{attribute addProperty BoxType "EK1100-0000-0018"}
{attribute addProperty Id "Beckhoff_EP9xxxEK1122Beckhoff_EP9xxxEK1122_D439D8FD4662582.75A_0023_EP9224_1037_0017EP9224_179A0949162A_0015_EP9128_2021_0019EP9128_179A0949162A_0014_EP9128_1021_0019EP9128_179A0949162A_0012_EP9128_2021_0018EP9128_179A0949162A_0011_EP9128_1021_0018EP9128_179A0949162A_0009_EP9128_2021_0017EP9128_179A0949162A_0008_EP9128_1021_0017EP9128_179A0949162A_0006_EP9128_2021_0016EP9128_179A0949162A_0005_EP9128_1021_0016EP9128_179A0949162A_0003_EP9128_2020_0016EP9128_179A0949162A_0002_EP9128_1020_0016EP9128_179A0949162"}
{attribute addProperty CRC "1080266710"}
{attribute addProperty SizeInBites "4838"}
{attribute addProperty SizeInBytes "604.75"}
TYPE Beckhoff_EP9xxx_40638FD6 EXTENDS EK1100_179A0949 :
STRUCT
	{attribute addProperty Name "Beckhoff_EP9xxxEK1122"}
	Beckhoff_EP9xxxEK1122 : Beckhoff_EP9xxxEK1122_D439D8FD;
	{attribute addProperty Name "A_0023_EP9224_1037_0017"}
	A_0023_EP9224_1037_0017 : EP9224_179A0949;
	{attribute addProperty Name "A_0015_EP9128_2021_0019"}
	A_0015_EP9128_2021_0019 : EP9128_179A0949;
	{attribute addProperty Name "A_0014_EP9128_1021_0019"}
	A_0014_EP9128_1021_0019 : EP9128_179A0949;
	{attribute addProperty Name "A_0012_EP9128_2021_0018"}
	A_0012_EP9128_2021_0018 : EP9128_179A0949;
	{attribute addProperty Name "A_0011_EP9128_1021_0018"}
	A_0011_EP9128_1021_0018 : EP9128_179A0949;
	{attribute addProperty Name "A_0009_EP9128_2021_0017"}
	A_0009_EP9128_2021_0017 : EP9128_179A0949;
	{attribute addProperty Name "A_0008_EP9128_1021_0017"}
	A_0008_EP9128_1021_0017 : EP9128_179A0949;
	{attribute addProperty Name "A_0006_EP9128_2021_0016"}
	A_0006_EP9128_2021_0016 : EP9128_179A0949;
	{attribute addProperty Name "A_0005_EP9128_1021_0016"}
	A_0005_EP9128_1021_0016 : EP9128_179A0949;
	{attribute addProperty Name "A_0003_EP9128_2020_0016"}
	A_0003_EP9128_2020_0016 : EP9128_179A0949;
	{attribute addProperty Name "A_0002_EP9128_1020_0016"}
	A_0002_EP9128_1020_0016 : EP9128_179A0949;
END_STRUCT
END_TYPE

(* stored: Version 1.2.0.0, ProductVersion 3.1.4024.9
   DUT Beckhoff_EP9xxx_40638FD6: Id {3be56f2e-639e-4ebb-b368-54025d46c849} *)
